FUNCTION_BLOCK FB_PPM_States
VAR_IN_OUT
    stMotionStage: DUT_MotionStage;
END_VAR
VAR_INPUT
    bEnable: BOOL;
    {attribute 'pytmc' := '
        pv: SET
        io: io
    '}
    enumSet: ENUM_PPM_states;
    bStatesLock: BOOL;
    fOut: LREAL;
    fPower: LREAL;
    fPolished: LREAL;
    fFrosted: LREAL;
END_VAR
VAR_OUTPUT
    bError: BOOL;
    sErrorMessage: STRING;
    bBusy: BOOL;
    bDone: BOOL;
    {attribute 'pytmc' := '
        pv: GET
        io: i
    '}
    enumGet: ENUM_PPM_States;
END_VAR
VAR
    bInit: BOOL;
    arrStates: ARRAY[1..15] OF DUT_PositionState;
    nIter: INT;

    {attribute 'pytmc' := '
        pv:
        io: io
    '}
    fbStateManager: FB_PositionStateManager;

    fbLockOut: FB_PositionStateLock;
    fbLockPowerMeter: FB_PositionStateLock;
    fbLockPolishedYag: FB_PositionStateLock;
    fbLockFrostedYag: FB_PositionStateLock;
END_VAR
VAR CONSTANT
    fInDelta: LREAL := 0.1;
    fOutDelta: LREAL := 10;
    fInVelocity: LREAL := 65;
    fOutVelocity: LREAL := 65;
    fAccel: LREAL := 1000;
    fOutDecel: LREAL := 1000;
END_VAR

IF NOT bInit THEN
    bInit := FALSE;
    FOR nIter := 1 TO 4 DO
        arrStates[nIter].fDelta := fInDelta;
        arrStates[nIter].fVelocity := fInVelocity;
        arrStates[nIter].fAccel := fAccel;
        arrStates[nIter].fDecel := fAccel;
        arrStates[nIter].bLocked := bStatesLock;
        arrStates[nIter].bValid := TRUE;
        // TODO implement PMPS instead of doing this
        arrStates[nIter].bMoveOk := TRUE;
    END_FOR
    arrStates[1].sName := 'Out';
    arrStates[1].fPosition := fOut;
    arrStates[1].fDelta := fOutDelta;
    arrStates[1].fVelocity := fOutVelocity;
    arrStates[1].fDecel := fOutDecel;
    arrStates[2].sName := 'PowerMeter';
    arrStates[2].fPosition := fPower;
    arrStates[3].sName := 'PolishedYag';
    arrStates[3].fPosition := fPolished;
    arrStates[4].sName := 'FrostedYag';
    arrStates[4].fPosition := fFrosted;
END_IF

fbLockOut(stPositionState := arrStates[1]);
fbLockPowerMeter(stPositionState := arrStates[2]);
fbLockPolishedYag(stPositionState := arrStates[3]);
fbLockFrostedYag(stPositionState := arrStates[4]);

fbStateManager(
    stMotionStage := stMotionStage,
    arrStates := arrStates,
    setState := enumSet,
    bEnable := bEnable,
    bError => bError,
    sErrorMessage => sErrorMessage,
    bBusy => bBusy,
    bDone => bDone,
    getState => enumGet);

END_FUNCTION_BLOCK

(* stored: Version 1.1.0.1, ProductVersion 3.1.4022.18
   POU FB_PPM_States: Id {1eb578bc-c89e-4a7a-b190-99dc56373dc2}, SpecialFunc None *)
